FUNCTION_BLOCK FB_DifferentCVCamera EXTENDS FB_ActionBasic
VAR_INPUT
    xExecute    : BOOL;
    xAbort      : BOOL;
	xReset		: BOOL;
    Cylinder 	: REFERENCE TO UNI_CylinderList;
    TimeOut  	: LREAL := 600; // Unit : s
	Input		: ST_InputTable;
	OutPut		: ST_OutputTable;
	Motor		: REFERENCE TO UNI_MotorList;
	BoxCameraDone :BOOL;
END_VAR	
VAR_OUTPUT
    xAborted : BOOL;
    iErrorID : INT;
    ErrorMsg : STRING;
	UseBoxCamera	:BOOL;
END_VAR
VAR
    StateBehaviour   : CBML.ETrigATo;
    CurrentPosition : ST_PositionTable;
	uiCyclicStep    : UINT := 0;
	TON_DelaySensor	:TON;
	TON_TimeOut		:TON;
	TON_ArriviedTimeOut :TON ;
	TON_CameraTimeOut	:TON;
	TON_ConveyorTimeOut	:TON;
	Reset_Rtrig 	:R_TRIG;
	fbExecuteEdgeDetect :FB_EdgeDetect;
	// ========== Resume 續做機制 ==========
	uiResumeStep	: UINT := 0;		// 錯誤發生時記錄的步驟，供續做使用
	bResumeEnabled	: BOOL := FALSE;	// 續做模式啟用旗標
END_VAR

THIS^.IBehaviourModel := StateBehaviour;
StateBehaviour(xExecute := xExecute,
              xAbort := xAbort OR fbExecuteEdgeDetect.xFallingEdge,
              udiTimeOut := LREAL_TO_UDINT( TimeOut*1000000),
              xDone => xDone,
              xBusy => xBusy,
              xError => xError,
              xAborted => xAborted);

iErrorID := StateBehaviour._model.iErrorID;
ErrorMsg := M_GetErrorMsg(xErrorID := iErrorID);

fbExecuteEdgeDetect(xInput :=xExecute);

Reset_Rtrig(CLK:= xReset);
IF Reset_Rtrig.Q THEN
	StateBehaviour.ResetModel(xCommit:=xReset);
END_IF

A00_BaseUnits();

ACTION A00_BaseUnits:
TON_DelaySensor(PT:= T#1S);
TON_TimeOut(PT := T#20S);
TON_ArriviedTimeOut(PT:= T#60S);
TON_CameraTimeOut(PT :=T#250S);
TON_ConveyorTimeOut(PT :=T#60S);
END_ACTION

METHOD CleanupAction
VAR_INPUT
    xAbortProposed : BOOL;
    iErrorIDProposed: INT;
END_VAR
VAR_OUTPUT
    xComplete : BOOL := TRUE;
    xAbort: BOOL := xAbortProposed;
 	iErrorID : INT := iErrorIDProposed;
END_VAR
xComplete := FALSE;

// ============================================================
// Resume 機制：保存當前步驟供後續 Resume 使用
// ============================================================
IF uiResumeStep = 0 THEN
	uiResumeStep := uiCyclicStep;
END_IF

// 清除所有 Timer
TON_DelaySensor.IN 		:= FALSE;
TON_TimeOut.IN 			:= FALSE;
TON_ArriviedTimeOut.IN 	:= FALSE;
TON_CameraTimeOut.IN 	:= FALSE;
TON_ConveyorTimeOut.IN 	:= FALSE;

// 重置輸出信號
UseBoxCamera 	:= FALSE;
BoxCameraDone 	:= FALSE;

// 機械復位到安全狀態
IF NOT xExecute THEN 
	Cylinder.List.fbDifferentSizeCV_Block1.M_Retract();
END_IF
Motor.List.TransmitDifferentSideCV.M_MotorStop();

// 等待機械復位完成
IF NOT xExecute THEN
	IF Cylinder.List.fbDifferentSizeCV_Block1.InRearPosition AND
	   Motor.List.TransmitDifferentSideCV.InStopped THEN
		xComplete := TRUE;
	END_IF
ELSE	
	IF Motor.List.TransmitDifferentSideCV.InStopped THEN
		xComplete := TRUE;
	END_IF
END_IF
END_METHOD

METHOD CyclicAction
VAR_INPUT
    itfTimingController : CBML.ITimingController;
END_VAR
VAR_OUTPUT
    xComplete : BOOL := TRUE;
    iErrorID : INT := 0;
END_VAR
VAR_INST
	bMoveConveyorForward	 : BOOL;
END_VAR
xComplete := FALSE;
IF bMoveConveyorForward THEN
	IF NOT Motor.List.TransmitDifferentSideCV.InBackWard THEN
		Motor.List.TransmitDifferentSideCV.M_MoveForward();
	END_IF
END_IF
CASE uiCyclicStep OF
	0:	// 初始化
		bMoveConveyorForward:=FALSE;
		uiCyclicStep :=1000;
		
	1000:	// 擋第一個盒子
		TON_TimeOut.IN:=TRUE;
		Cylinder.List.fbDifferentSizeCV_Block1.M_Extend();
		Cylinder.List.fbTransmitCV_CamaraHoriz.M_Extend();
		IF Cylinder.List.fbDifferentSizeCV_Block1.InFrontPosition AND
			Cylinder.List.fbTransmitCV_CamaraHoriz.InFrontPosition THEN
			TON_TimeOut.IN:=FALSE;
			uiCyclicStep :=1050;
		END_IF
		IF TON_TimeOut.Q THEN
			uiResumeStep := uiCyclicStep;
			iErrorID := 7;
		END_IF

	1050:	// 馬達前進
		TON_ConveyorTimeOut.IN:=TRUE;
		bMoveConveyorForward:=TRUE;
		Cylinder.List.fbDifferentSizeCV_Press1.M_Retract();
		IF Motor.List.TransmitDifferentSideCV.InForWard AND
			Cylinder.List.fbDifferentSizeCV_Press1.InRearPosition THEN
			TON_ConveyorTimeOut.IN:= FALSE;
			uiCyclicStep :=1100;
		END_IF
		IF TON_ConveyorTimeOut.Q THEN
			uiResumeStep := uiCyclicStep;
			iErrorID := 7;
		END_IF

	1100:	// 檢查盒子到達擋塊
		TON_ArriviedTimeOut.IN:=TRUE;
		TON_DelaySensor.IN:=Input.bDifferentSizeCV_BoxDetect2_Sensor;
		IF TON_DelaySensor.Q THEN
			TON_DelaySensor.IN :=FALSE;
			TON_ArriviedTimeOut.IN :=FALSE;
			Cylinder.List.fbDifferentSizeCV_Press1.M_Extend();
			bMoveConveyorForward:=FALSE;
			Motor.List.TransmitDifferentSideCV.M_MotorStop();
			uiCyclicStep :=1200;
		END_IF
		IF TON_ArriviedTimeOut.Q THEN
			uiResumeStep := uiCyclicStep;
			iErrorID := 8;
		END_IF

	1200:	// 發送拍照請求 & 擋住第二個盒子
		TON_ConveyorTimeOut.IN:=TRUE;
		IF Cylinder.List.fbDifferentSizeCV_Press1.InFrontPosition AND
			Motor.List.TransmitDifferentSideCV.InStopped THEN
			TON_ConveyorTimeOut.IN:= FALSE;
			UseBoxCamera :=TRUE;
			uiCyclicStep :=1300;
		END_IF
		IF TON_ConveyorTimeOut.Q THEN
			uiResumeStep := uiCyclicStep;
			iErrorID := 9;
		END_IF

	1300:	// 等待 C# 拍照完成 (Camera 錯誤不可續做)
		TON_CameraTimeOut.IN:=TRUE;
		IF BoxCameraDone THEN
			TON_CameraTimeOut.IN :=FALSE;
			Cylinder.List.fbDifferentSizeCV_Block1.M_Retract();
			bMoveConveyorForward:=TRUE;
			uiCyclicStep :=1400;
		END_IF
		IF TON_CameraTimeOut.Q THEN
			uiResumeStep := uiCyclicStep;
			iErrorID :=10;
		END_IF

	1400:	// 盒子通過 Detect1 感測器
		TON_TimeOut.IN :=TRUE;
		IF Input.bDifferentSizeCV_BoxDetect1_Sensor THEN
			TON_TimeOut.IN :=FALSE;
			uiCyclicStep :=1500;
		END_IF
		IF TON_TimeOut.Q THEN
			uiResumeStep := uiCyclicStep;
			iErrorID :=11;
		END_IF

	1500:	// 離開感測器後停止馬達
		TON_DelaySensor.IN:=TRUE;
		IF NOT Input.bDifferentSizeCV_BoxDetect1_Sensor THEN
			TON_DelaySensor.IN:=FALSE;
			bMoveConveyorForward:=FALSE;
			Motor.List.TransmitDifferentSideCV.M_MotorStop();
			uiCyclicStep :=1600;
		END_IF
		IF TON_DelaySensor.Q THEN
			TON_DelaySensor.IN:=FALSE;
			bMoveConveyorForward:=FALSE;
			Motor.List.TransmitDifferentSideCV.M_MotorStop();
			uiCyclicStep :=1600;
		END_IF
	
	1600:	// 等待馬達停止
		IF Motor.List.TransmitDifferentSideCV.InStopped THEN
			xComplete :=TRUE;
		END_IF

END_CASE
END_METHOD

METHOD ExitAction
VAR_INPUT
    xAfterCleanup : BOOL;
    xInCopyCode : BOOL;
END_VAR
END_METHOD

METHOD M_GetErrorMsg : T_MaxString
VAR_INPUT
	xErrorID: INT;
END_VAR

VAR
	
END_VAR
CASE xErrorID OF
	0:
		M_GetErrorMsg := 'No Error';
	1:
		M_GetErrorMsg := 'Action time out';
	2:
		M_GetErrorMsg := 'Position Data invalid';
	3:
		M_GetErrorMsg := 'Block1 cylinder not ready';
	4:
		M_GetErrorMsg := 'Press1 cylinder not ready';
	5:
		M_GetErrorMsg := 'CamaraHoriz cylinder not ready';
	6:
		M_GetErrorMsg := 'DifferentCV not ready ';
	7:
		M_GetErrorMsg := 'Cylinder timeout';
	8:
		M_GetErrorMsg :='photo area have not box timeout';
	9:
		M_GetErrorMsg :='motor & cylinder timeout';
	10:
		M_GetErrorMsg :='C# BoxCameraDone timeout';
	11:
		M_GetErrorMsg :='Box cross sensor not detact timeout';
		
	20:
		M_GetErrorMsg :='Differnet conveyor full box infront';
END_CASE
END_METHOD

METHOD ResetAction
VAR_OUTPUT
    xComplete : BOOL := TRUE;
END_VAR
xComplete := FALSE;

// ============================================================
// Resume 機制判斷
// ------------------------------------------------------------
// 當錯誤發生後，操作員可選擇：
//   1. 保持 xExecute = TRUE 並按 Reset → Resume (從錯誤點繼續)
//   2. 先關閉 xExecute，再重新啟動 → 從頭開始
// ============================================================
bResumeEnabled := xExecute;

// 如果不是 Resume 模式，清除 Resume 步驟記錄
IF NOT bResumeEnabled THEN
	uiResumeStep := 0;
END_IF

// 清除所有 Timer
TON_DelaySensor.IN 		:= FALSE;
TON_TimeOut.IN 			:= FALSE;
TON_ArriviedTimeOut.IN 	:= FALSE;
TON_CameraTimeOut.IN 	:= FALSE;
TON_ConveyorTimeOut.IN 	:= FALSE;

xComplete := TRUE;
END_METHOD

METHOD StartAction
VAR_OUTPUT
    xComplete : BOOL := TRUE;
	iErrorID : INT := 0;
END_VAR
VAR
	bIsResumeMode : BOOL;	// 局部變數：記錄是否為 Resume 模式
END_VAR
xComplete := FALSE;

// 清除所有 Timer
TON_DelaySensor.IN 		:= FALSE;
TON_TimeOut.IN 			:= FALSE;
TON_ArriviedTimeOut.IN 	:= FALSE;
TON_CameraTimeOut.IN 	:= FALSE;
TON_ConveyorTimeOut.IN 	:= FALSE;

// ============================================================
// Resume 機制處理
// ------------------------------------------------------------
// 可 Resume 的錯誤: Error 7, 8, 9, 11 (氣缸/馬達/等待盒子)
// 不可 Resume 的錯誤: Error 10 (C# 拍照失敗), Error 20 (輸送帶滿載)
// ============================================================
bIsResumeMode := bResumeEnabled AND uiResumeStep > 0 AND uiResumeStep <> 1300;

IF bResumeEnabled AND uiResumeStep > 0 THEN
	IF uiResumeStep = 1300 THEN
		// Camera 錯誤：不可 Resume，強制從頭開始
		uiCyclicStep 	:= 0;
		UseBoxCamera 	:= FALSE;
		BoxCameraDone 	:= FALSE;
	ELSE
		// 其他錯誤：允許 Resume (人工已確認可繼續)
		uiCyclicStep := uiResumeStep;
	END_IF
	// 清除 Resume 旗標
	bResumeEnabled 	:= FALSE;
	uiResumeStep 	:= 0;
ELSE
	// 正常模式：從頭開始
	uiCyclicStep 	:= 0;
	UseBoxCamera 	:= FALSE;
	BoxCameraDone 	:= FALSE;
END_IF

// ============================================================
// 啟動前錯誤檢查
// ============================================================
IF Input.bDifferentSizeCV_BoxDetect1_Sensor THEN
	iErrorID := 20;
END_IF

IF Cylinder.List.fbDifferentSizeCV_Block1.xError THEN
	iErrorID := 3;
END_IF
IF Cylinder.List.fbDifferentSizeCV_Press1.xError THEN
	iErrorID := 4;
END_IF
IF Cylinder.List.fbTransmitCV_CamaraHoriz.xError THEN
	iErrorID := 5;
END_IF
IF Motor.List.TransmitDifferentSideCV.xError THEN
	iErrorID := 6;
END_IF

// 完成條件：Resume 模式直接完成，正常模式需檢查初始位置
IF bIsResumeMode OR
   (Cylinder.List.fbDifferentSizeCV_Block1.InRearPosition AND
    Motor.List.TransmitDifferentSideCV.InStopped) THEN
	xComplete := TRUE;
END_IF
END_METHOD

END_FUNCTION_BLOCK

(* stored: Version 1.1.0.1, ProductVersion 3.1.4024.13
   POU FB_DifferentCVCamera: Id {f4ab733a-15a9-490a-bf47-b810290f7ccc}, SpecialFunc None
   Folder Action: Id {50b7549f-3c45-4ccf-a4a7-1cdf3c96151f}
   Action A00_BaseUnits: Id {ecb63a04-5545-4c1d-8290-f4ae59068027}
   Method CleanupAction: Id {84d205e3-84a9-4e6e-91e2-34f7af845f9a}
   Method CyclicAction: Id {dd093b31-2fe3-4187-9bd9-74b44ab660f6}
   Method ExitAction: Id {249c6dab-8479-4fb7-ad51-11e60e594e10}
   Method M_GetErrorMsg: Id {07171412-48bc-4271-a493-d60c93b6db04}
   Method ResetAction: Id {bbc4d767-cb94-4960-954c-a81bc8ad836f}
   Method StartAction: Id {d5f673ab-d024-4521-94fc-f22c207174d7} *)
